FUNCTION_BLOCK FB_BaseStation IMPLEMENTS I_WorkingStation
VAR_INPUT
END_VAR
VAR_OUTPUT
END_VAR
VAR
	bRotationInterlock: BOOL;
	bRotationRequest: BOOL;
	fbTablePlace: REFERENCE TO FB_TablePlace;
	bError: BOOL;
	udiErrorNumber:UDINT;
	bTableInPosition: BOOL;
	bManualMode: BOOL;
	iWorkStep: INT;
END_VAR

METHOD mError : BOOL
VAR_INPUT
	udiErrorNumberSet: UDINT;
END_VAR
udiErrorNumber := udiErrorNumberSet;
bError := TRUE;
iWorkStep:=90;
END_METHOD

METHOD mErrorReset : BOOL
VAR_INPUT
END_VAR
bError := FALSE;
udiErrorNumber := 0;
iWorkStep:=91;
END_METHOD

PROPERTY pError : BOOL
GET
pError := bError;
END_GET
END_PROPERTY

PROPERTY pErrorNumber : UDINT
GET
pErrorNumber:= udiErrorNumber;
END_GET
END_PROPERTY

{attribute 'monitoring' := 'call'}
PROPERTY prTableInPosition : BOOL
GET
prTableInPosition:=bTableInPosition;
END_GET
SET
bTableInPosition:=prTableInPosition;
END_SET
END_PROPERTY

{attribute 'monitoring' := 'call'}
PROPERTY prTableRotationInterlock : BOOL
GET
prTableRotationInterlock := bRotationInterlock;
END_GET
SET
bRotationInterlock := prTableRotationInterlock;
END_SET
END_PROPERTY

{attribute 'monitoring' := 'call'}
PROPERTY prTableRotationRequest : BOOL
GET
prTableRotationRequest:= bRotationRequest;
END_GET
END_PROPERTY

PROPERTY pTablePlace : REFERENCE TO FB_TablePlace
GET
pTablePlace REF= fbTablePlace;
END_GET
SET
fbTablePlace REF= pTablePlace;
END_SET
END_PROPERTY

END_FUNCTION_BLOCK

(* stored: Version 1.1.0.1, ProductVersion 3.1.4024.15
   POU FB_BaseStation: Id {9cbe06d4-36ed-4e19-8636-f06f6ed53125}, SpecialFunc None
   Method mError: Id {fb83016a-aaa2-4dd7-8f9c-2795ee415507}
   Method mErrorReset: Id {307c245a-308f-4b3e-a89f-a5e87dd8cc62}
   Property pError: Id {b0d60995-960d-478b-b068-43a1eebae1e8}
   Get Get: Id {9f3de2f4-5df4-435d-80fb-a907e1adb63f}
   Property pErrorNumber: Id {d80a4a1f-6932-4311-bb5a-0f21cc367d92}
   Get Get: Id {062d2237-59a2-40b7-81f2-ad808ac10adf}
   Property prTableInPosition: Id {592cf85c-3254-4812-b020-5d141833f6ab}
   Get Get: Id {217c66a4-f5be-4f35-b16e-a6b86af79b22}
   Set Set: Id {bb7ede60-fba5-4c19-8c00-ebcefea92104}
   Property prTableRotationInterlock: Id {e5fc254a-5609-4be3-84a7-f8c244dac0b1}
   Get Get: Id {b7a6cd8a-205a-4ef0-80ee-061e503f9f54}
   Set Set: Id {dd4a82e4-3071-4331-955b-6cba30b3edf6}
   Property prTableRotationRequest: Id {4f6b0926-f186-40fb-a73a-e615918a2a53}
   Get Get: Id {e1c3145f-d20b-41e6-89c1-66bdfe48409e}
   Property pTablePlace: Id {88cbe737-a470-4003-9fa4-38b67688cbaf}
   Get Get: Id {bd357123-069c-4d22-9e1c-de08e6b4f1bb}
   Set Set: Id {17bc3b84-08fa-40ff-9713-9439282169b2} *)
